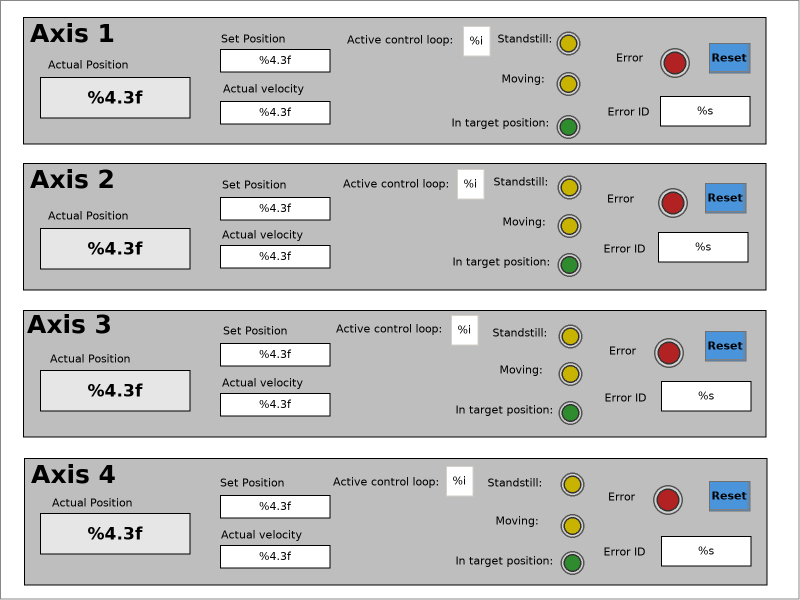
VISUALIZATION Screen1  // 800x600
    Rectangle (23,17 743x127)
    Rectangle (23,163 743x127)
    Rectangle (23,310 743x127)
    Rectangle (24,458 743x127)
    Label (27,18 110x30), "Axis 1"
    Label (27,164 110x30), "Axis 2"
    Label (24,309 110x30), "Axis 3"
    Label (28,459 110x30), "Axis 4"
    Textfield (40,77 150x41), "%4.3f", text variable: MAIN.Axis[0][MAIN.Axis1LoopID].NcToPlc.ActPos
    Label (45,50 150x30), "Actual Position"
    Label (45,201 150x30), "Actual Position"
    Label (47,344 150x30), "Actual Position"
    Label (49,488 150x30), "Actual Position"
    Textfield (40,228 150x41), "%4.3f", text variable: MAIN.Axis[1][MAIN.Axis2LoopID].NcToPlc.ActPos
    Textfield (40,370 150x41), "%4.3f", text variable: MAIN.Axis[2][MAIN.Axis3LoopID].NcToPlc.ActPos
    Textfield (40,513 150x41), "%4.3f", text variable: MAIN.Axis[3][MAIN.Axis4LoopID].NcToPlc.ActPos
    Label (218,24 150x30), "Set Position"
    Lamp1 (658,42 34x42), variable: MAIN.Axis[0][MAIN.Axis1LoopID].Status.Error, style: Lamp-Lamp1-Red
    Label (610,43 39x30), "Error"
    Label (596,97 65x30), "Error ID"
    Textfield (660,96 90x30), "%s", text variable: MAIN.Axis[0][MAIN.Axis1LoopID].Status.ErrorID
    Textfield (220,49 110x23), "%4.3f", text variable: MAIN.Axis[0][MAIN.Axis1LoopID].NcToPlc.TargetPos
    Textfield (220,101 110x23), "%4.3f", text variable: MAIN.Axis[0][MAIN.Axis1LoopID].NcToPlc.ActVelo
    Label (220,74 150x30), "Actual velocity"
    Label (219,170 150x30), "Set Position"
    Label (220,316 150x30), "Set Position"
    Label (217,468 150x30), "Set Position"
    Textfield (220,197 110x23), "%4.3f", text variable: MAIN.Axis[1][MAIN.Axis2LoopID].NcToPlc.TargetPos
    Textfield (220,343 110x23), "%4.3f", text variable: MAIN.Axis[2][MAIN.Axis3LoopID].NcToPlc.TargetPos
    Textfield (220,495 110x23), "%4.3f", text variable: MAIN.Axis[3][MAIN.Axis4LoopID].NcToPlc.TargetPos
    Label (219,220 150x30), "Actual velocity"
    Label (219,368 150x30), "Actual velocity"
    Label (218,520 150x30), "Actual velocity"
    Textfield (220,245 110x23), "%4.3f", text variable: MAIN.Axis[1][MAIN.Axis2LoopID].NcToPlc.ActVelo
    Textfield (220,393 110x23), "%4.3f", text variable: MAIN.Axis[3][MAIN.Axis3LoopID].NcToPlc.ActVelo
    Textfield (220,545 110x23), "%4.3f", text variable: MAIN.Axis[3][MAIN.Axis4LoopID].NcToPlc.ActVelo
    Label (601,184 39x30), "Error"
    Label (603,336 39x30), "Error"
    Label (602,482 39x30), "Error"
    Lamp1 (656,182 34x42), variable: MAIN.Axis[1][MAIN.Axis2LoopID].Status.Error, style: Lamp-Lamp1-Red
    Lamp1 (652,332 34x42), variable: MAIN.Axis[2][MAIN.Axis3LoopID].Status.Error, style: Lamp-Lamp1-Red
    Lamp1 (651,479 34x42), variable: MAIN.Axis[3][MAIN.Axis4LoopID].Status.Error, style: Lamp-Lamp1-Red
    Label (592,234 65x30), "Error ID"
    Label (593,383 65x30), "Error ID"
    Label (592,537 65x30), "Error ID"
    Textfield (658,232 90x30), "%s", text variable: MAIN.Axis[1][MAIN.Axis2LoopID].Status.ErrorID
    Textfield (661,381 90x30), "%s", text variable: MAIN.Axis[2][MAIN.Axis3LoopID].Status.ErrorID
    Textfield (661,536 90x30), "%s", text variable: MAIN.Axis[3][MAIN.Axis4LoopID].Status.ErrorID
    Lamp1 (555,67 27x34), variable: MAIN.Axis[0][MAIN.Axis1LoopID].Status.Moving, style: Lamp-Lamp1-Yellow
    Lamp1 (555,110 27x34), variable: MAIN.Axis[0][MAIN.Axis1LoopID].Status.InTargetPosition, style: Lamp-Lamp1-Green
    Label (491,24 68x30), "Standstill:"
    Label (450,108 101x30), "In target position:"
    Lamp1 (555,26 27x35), variable: MAIN.Axis[0][MAIN.Axis1LoopID].Status.StandStill, style: Lamp-Lamp1-Yellow
    Label (490,207 68x30), "Moving:"
    Lamp1 (556,170 27x35), variable: MAIN.Axis[1][MAIN.Axis2LoopID].Status.StandStill, style: Lamp-Lamp1-Yellow
    Lamp1 (556,209 27x34), variable: MAIN.Axis[1][MAIN.Axis2LoopID].Status.Moving, style: Lamp-Lamp1-Yellow
    Lamp1 (556,248 27x34), variable: MAIN.Axis[1][MAIN.Axis2LoopID].Status.InTargetPosition, style: Lamp-Lamp1-Green
    Lamp1 (559,467 27x35), variable: MAIN.Axis[3][MAIN.Axis4LoopID].Status.StandStill, style: Lamp-Lamp1-Yellow
    Lamp1 (557,319 27x35), variable: MAIN.Axis[2][MAIN.Axis3LoopID].Status.StandStill, style: Lamp-Lamp1-Yellow
    Lamp1 (557,357 27x34), variable: MAIN.Axis[2][MAIN.Axis3LoopID].Status.Moving, style: Lamp-Lamp1-Yellow
    Lamp1 (559,509 27x34), variable: MAIN.Axis[3][MAIN.Axis4LoopID].Status.Moving, style: Lamp-Lamp1-Yellow
    Lamp1 (557,396 27x34), variable: MAIN.Axis[2][MAIN.Axis3LoopID].Status.InTargetPosition, style: Lamp-Lamp1-Green
    Lamp1 (559,546 27x34), variable: MAIN.Axis[3][MAIN.Axis4LoopID].Status.InTargetPosition, style: Lamp-Lamp1-Green
    Label (487,167 68x30), "Standstill:"
    Label (486,318 68x30), "Standstill:"
    Label (481,468 68x30), "Standstill:"
    Label (489,64 68x30), "Moving:"
    Label (487,355 68x30), "Moving:"
    Label (483,506 68x30), "Moving:"
    Label (451,247 101x30), "In target position:"
    Label (454,395 101x30), "In target position:"
    Label (454,546 101x30), "In target position:"
    Label (342,25 116x30), "Active control loop:"
    Textfield (463,26 27x30), "%i", text variable: MAIN.Axis[0][0].NcToPlc.ActiveControlLoopIndex
    Textfield (457,169 27x30), "%i", text variable: MAIN.Axis[1][0].NcToPlc.ActiveControlLoopIndex
    Textfield (451,315 27x30), "%i", text variable: MAIN.Axis[2][0].NcToPlc.ActiveControlLoopIndex
    Textfield (446,466 27x30), "%i", text variable: MAIN.Axis[3][0].NcToPlc.ActiveControlLoopIndex
    Label (338,169 116x30), "Active control loop:"
    Label (331,314 116x30), "Active control loop:"
    Label (328,467 116x30), "Active control loop:"
    Button (709,43 41x30), "Reset"
        OnMouseDown: execute { MAIN.Reset(Axis:=MAIN.Axis[0][MAIN.Axis1LoopID],Execute:=TRUE); MAIN.Reset(Axis:=MAIN.Axis[0][MAIN.Axis1LoopID],Execute:=FALSE); }
    Button (705,183 41x30), "Reset"
        OnMouseDown: execute { MAIN.Reset(Axis:=MAIN.Axis[1][MAIN.Axis2LoopID],Execute:=TRUE); MAIN.Reset(Axis:=MAIN.Axis[1][MAIN.Axis2LoopID],Execute:=FALSE); }
    Button (705,331 41x30), "Reset"
        OnMouseDown: execute { MAIN.Reset(Axis:=MAIN.Axis[2][MAIN.Axis3LoopID],Execute:=TRUE); MAIN.Reset(Axis:=MAIN.Axis[2][MAIN.Axis3LoopID],Execute:=FALSE); }
    Button (709,481 41x30), "Reset"
        OnMouseDown: execute { MAIN.Reset(Axis:=MAIN.Axis[3][MAIN.Axis4LoopID],Execute:=TRUE); MAIN.Reset(Axis:=MAIN.Axis[3][MAIN.Axis4LoopID],Execute:=FALSE); }
END_VISUALIZATION

(* stored: Version 1.1.0.1, ProductVersion 3.1.4024.12
   Visu Screen1: Id {cc69c11d-d32d-4f5d-a295-2cea608d6771} *)
